TYPE ST_GROUP_INFO :
STRUCT
  GroupStatusValid,
  GroupStatusBusy,
  GroupMoving, 
  GroupHoming, 
  GroupErrorStop, 
  GroupNotReady, 
  GroupStandby, 
  GroupStopping,
 
  GroupDisabled, 
  AllAxesStanding, 
  ConstantVelocity, 
  Accelerating, 
  Decelerating, 
  InPosition, 
  GroupError					: BIT; 

  GroupErrorId					: UDINT;

   AxisCount      				: UDINT;
END_STRUCT
END_TYPE

(* stored: Version 1.1.0.1, ProductVersion 3.1.4024.12
   DUT ST_GROUP_INFO: Id {fa1bc841-4934-459e-882e-2c7e4af57157} *)
